Yaskawa INFORM job: X2_99(90,0).JBI

/JOB
//NAME X2_99(90,0)
///FOLDERNAME X2
//POS
///NPOS 440,440,436,13,0,0
///TOOL 0
///POSTYPE PULSE
///PULSE
C00000=2000,-99612,-82443,0,53832,0
C00001=-166393,-132062,-92618,58483,55149,81008
C00002=-157482,-99612,-82443,50725,53832,-76817
C00003=-152781,-96239,-78741,49340,50884,-75750
C00004=-150954,-94792,-77210,48744,49760,-75306
C00005=-150957,-94045,-75225,49281,49201,-75681
C00006=-151067,-94769,-77060,48840,49767,-75375
C00007=-148896,-96259,-77631,48213,48319,-74911
C00008=-154925,-106114,-81211,52368,49780,-77962
C00009=-154976,-104737,-78409,53070,49177,-78455
C00010=-153765,-101609,-77307,52041,49068,-77683
C00011=-154727,-103781,-80113,51957,49998,-77663
C00012=-157482,-99612,-82443,50725,53832,-76817
C00013=-126812,-81448,-90767,9472,77282,-14340
C00014=-120783,-85892,-98127,-47,82159,60
C00015=-120791,-78998,-92147,-45,82022,58
C00016=-120812,-59041,-81112,-38,85486,50
C00017=-120812,-59638,-79752,-38,84341,50
C00018=-120812,-59041,-81112,-38,85486,50
C00019=-120792,-70899,-87175,-45,83124,57
C00020=-120810,-72484,-85548,-40,81307,51
C00021=-120817,-76009,-87202,-37,80512,50
C00022=-120816,-72927,-85752,-37,81205,50
C00023=-120792,-71723,-87920,-45,83159,57
C00024=-120783,-85892,-98127,-47,82159,60
C00025=-120841,-86418,-98444,-30,82084,41
C00026=-120867,-62955,-84955,-21,85839,32
C00027=-120862,-57449,-80347,-23,85833,34
C00028=-120862,-58065,-78999,-24,84687,34
C00029=-120862,-57449,-80347,-23,85833,34
C00030=-120848,-76846,-90076,-28,81853,39
C00031=-120700,-77430,-87681,-72,80079,89
C00032=-120707,-73445,-85814,-70,80978,86
C00033=-120700,-77430,-87681,-72,80079,89
C00034=-120841,-86418,-98444,-30,82084,41
C00035=-120877,-85820,-98106,-19,82183,30
C00036=-120894,-60284,-82721,-14,85837,23
C00037=-120891,-57831,-80469,-15,85712,24
C00038=-120891,-58439,-79117,-15,84567,25
C00039=-120891,-57831,-80469,-15,85712,24
C00040=-120882,-76306,-89742,-18,81925,28
C00041=-120632,-76849,-87581,-92,80316,111
C00042=-120641,-72870,-85708,-89,81208,107
C00043=-120899,-105607,-111704,-13,80383,24
C00044=-120899,-105607,-111704,-13,80383,24
C00045=-120329,-64675,-84682,-181,84785,205
C00046=-120337,-61857,-81845,-179,84488,203
C00047=-120337,-62228,-80870,-179,83698,204
C00048=-120337,-61849,-81865,-179,84506,203
C00049=-120308,-72964,-87409,-188,82206,216
C00050=-112365,-66887,-81837,-2540,82030,2815
C00051=-112466,-65041,-80903,-2509,82400,2777
C00052=-112291,-68228,-82506,-2565,81755,2847
C00053=-88690,-37051,-64863,-22386,100281,29037
C00054=-90338,-32373,-60570,-22143,99643,28585
C00055=-86677,-30127,-56933,-28301,101078,28609
C00056=-87262,-30704,-57322,-28229,100840,28451
C00057=-86036,-30845,-57417,-28365,101220,28810
C00058=-80749,-50154,-73696,-28906,103010,30322
C00059=-106026,-92840,-102541,-4408,81700,4909
C00060=-104933,-21068,-63327,-14588,98299,15445
C00061=-118026,-7058,-59426,2478,121298,42537
C00062=-119206,-9959,-57512,2402,118662,42076
C00063=-119679,-11008,-56668,2374,117617,41892
C00064=-119678,-12040,-55711,2348,116499,41868
C00065=-119679,-11008,-56668,2374,117617,41892
C00066=-117888,-11929,-55575,2351,116426,42475
C00067=-118578,-11982,-55616,2350,116441,42241
C00068=-117888,-11929,-55575,2351,116426,42475
C00069=-116239,-8118,-58416,2447,120087,43116
C00070=-117941,-7017,-59404,2478,121303,42566
C00071=-119121,-9922,-57492,2402,118667,42105
C00072=-119594,-10972,-56650,2375,117622,41921
C00073=-119593,-12004,-55694,2348,116504,41897
C00074=-119594,-10972,-56650,2375,117622,41921
C00075=-117972,-11968,-55595,2351,116420,42446
C00076=-118663,-12020,-55635,2349,116436,42212
C00077=-117972,-11968,-55595,2351,116420,42446
C00078=-116323,-8162,-58441,2447,120082,43087
C00079=-118213,-4464,-57342,2479,121353,42475
C00080=-119375,-7335,-55445,2404,118742,42020
C00081=-119840,-8375,-54609,2376,117706,41839
C00082=-119839,-9401,-53662,2350,116597,41815
C00083=-119840,-8375,-54609,2376,117706,41839
C00084=-117787,-9255,-53494,2353,116516,42511
C00085=-118466,-9310,-53537,2352,116532,42281
C00086=-117787,-9255,-53494,2353,116516,42511
C00087=-113921,-56504,-90793,-659,90254,43086
C00088=-172997,-84117,-74043,29270,60841,12459
C00089=-182497,-62439,-47217,33561,35566,5540
C00090=-177866,51889,12751,25241,78726,20035
C00091=-177567,56483,20827,25353,76270,19609
C00092=-177451,58453,24226,25418,75255,19428
C00093=-177454,58193,25598,25524,74370,19231
C00094=-177460,58244,25401,25510,74505,19259
C00095=-177296,61431,29027,25518,73918,19189
C00096=-177460,58244,25401,25510,74505,19259
C00097=-177875,51523,13769,25307,77989,19872
C00098=-167005,53799,14731,23971,77323,24144
C00099=-166588,57735,22127,23390,74500,23603
C00100=-165356,57001,22663,20748,72181,23241
C00101=-165358,56731,24024,20856,71266,23076
C00102=-165347,56799,23771,20830,71442,23111
C00103=-165330,60004,27398,20889,70889,23018
C00104=-165347,56799,23771,20830,71442,23111
C00105=-166977,49436,12685,24253,74137,23502
C00106=-182364,4853,-37106,25072,86261,16971
C00107=-152303,-102933,-107906,-365,71882,21471
C00108=-90355,-25240,-62492,-31182,91940,-14489
C00109=-138081,35844,8180,-39695,66399,-31141
C00110=-138669,40694,16134,-40133,64268,-30541
C00111=-138897,42750,19469,-40345,63394,-30283
C00112=-138897,42781,21161,-40673,62603,-29947
C00113=-138886,42628,20611,-40593,62809,-30029
C00114=-139201,45623,23796,-40603,62339,-29981
C00115=-138886,42628,20611,-40593,62809,-30029
C00116=-138069,35590,9192,-39905,65818,-30900
C00117=-133067,14417,-5479,-38193,49171,-52584
C00118=-129431,19961,2498,-38515,39991,-63248
C00119=-130261,24926,10174,-39520,37911,-62617
C00120=-130583,27008,13377,-40001,37063,-62330
C00121=-130583,27275,15303,-40912,36255,-61820
C00122=-130584,27314,14967,-40710,36428,-61933
C00123=-131029,30096,17715,-40568,36020,-61996
C00124=-130584,27314,14967,-40710,36428,-61933
C00125=-124769,26347,15261,-56693,39526,-56291
C00126=-125951,31813,23350,-58329,37603,-55322
C00127=-125990,33793,23574,-57346,38066,-55879
C00128=-123661,25065,17775,-59577,38998,-54642
C00129=-125990,34597,27233,-59382,37066,-54726
C00130=-126486,36192,28495,-62823,42923,-46041
C00131=-130207,41845,28467,-57474,57413,-30842
C00132=-133480,44167,26403,-51334,63232,-25301
C00133=-133401,42077,23210,-51024,63850,-25633
C00134=-132439,36745,15005,-50531,65875,-26297
C00135=-90355,-25240,-62492,-31182,91940,-14489
C00136=-126181,-67140,-93758,-13250,84858,5822
C00137=-152303,-102933,-107906,-365,71882,21471
C00138=-151021,-50166,-89002,-846,87371,21807
C00139=-182364,4853,-37106,25072,86261,16971
C00140=-184325,60344,23585,34019,76352,15866
C00141=-183678,65674,32396,34159,73860,15344
C00142=-183957,81689,47427,34502,79595,16153
C00143=-184996,71033,34569,34595,82030,16501
C00144=-183957,81525,49351,34624,78541,15822
C00145=-167608,69842,33487,23377,75298,21262
C00146=-169419,57377,22961,28412,70050,19919
C00147=-169758,52135,14437,28170,72420,20393
C00148=-182364,4853,-37106,25072,86261,16971
C00149=-152303,-102933,-107906,-365,71882,21471
C00150=-121941,-117598,-112997,-12501,69917,32230
C00151=-108451,-171803,-109385,-23800,43994,42320
C00152=-115265,-105280,-99916,-13150,93342,30989
C00153=-112792,-107844,-97393,-16343,91026,32017
C00154=-122694,-143516,-106419,-10106,61697,32034
C00155=-122359,-107950,-95942,-9400,73404,31180
C00156=-122118,-61038,-75540,-9150,84839,30407
C00157=-121770,-8357,-41103,-9216,90729,30109
C00158=-121771,-1968,-35922,-9217,90821,30102
C00159=-121055,-283,-39052,-9429,93653,30116
C00160=-118931,-1420,-16721,-1449,102592,42361
C00161=-118945,163,-15392,-1659,93503,40633
C00162=-120171,930,-10959,-1582,91145,40250
C00163=-120660,1326,-9108,-1553,90200,40098
C00164=-120694,25865,13192,-1550,89085,40100
C00165=-120696,29026,16285,-1550,88805,40104
C00166=-120258,23290,9189,-1576,90234,40233
C00167=-119165,22386,4533,-1644,92655,40570
C00168=-119181,24192,6266,-1459,101602,42286
C00169=-120260,23811,9690,-1517,99280,41943
C00170=-120693,23749,11149,-1541,98342,41806
C00171=-120660,1326,-9108,-1544,99287,41805
C00172=-120174,1432,-10536,-1517,100229,41961
C00173=-118965,1918,-13913,-1451,102579,42349
C00174=-119164,21752,3941,-1459,101779,42290
C00175=-120255,21351,7351,-1518,99456,41942
C00176=-120694,21281,8802,-1542,98518,41803
C00177=-120641,1282,-9371,-1543,99426,41811
C00178=-120163,-1908,-13337,-1516,100237,41964
C00179=-118931,-1420,-16721,-1449,102592,42361
C00180=-109578,15420,-7310,-28367,110236,-41857
C00181=-109763,14188,-4345,-27924,107995,-41350
C00182=-110193,13805,-2890,-27787,106881,-41239
C00183=-131022,13378,-3260,-29129,99839,-47636
C00184=-122106,10683,8881,-53521,92538,-44133
C00185=-120623,10562,7326,-53535,93941,-44154
C00186=-119164,10594,3761,-53715,96134,-44669
C00187=-115308,-32515,-29810,-53374,97452,-43308
C00188=-160324,-56725,-62447,4686,86573,-10750
C00189=-150232,17988,-5017,26557,112251,35280
C00190=-142954,11495,-10959,27504,110227,37702
C00191=-142768,10690,-7556,27067,107926,37200
C00192=-143003,11007,-5424,26849,106972,36875
C00193=-137789,7639,-8393,27391,105376,38540
C00194=-140743,9596,5422,48538,102657,38323
C00195=-145934,20226,29397,62426,105383,26201
C00196=-142397,10029,6905,51885,103476,38119
C00197=-144627,12481,5478,52145,106089,38424
C00198=-150232,17988,-5017,26557,112251,35280
C00199=-160324,-56725,-62447,4686,86573,-10750
C00200=-146496,-53907,-57071,50358,82742,77471
C00201=-142086,-46087,-49611,49702,79955,78251
C00202=-140910,-47839,-49478,49629,78666,78171
C00203=-141016,-46873,-48908,49627,78820,78198
C00204=-140042,-41059,-45363,49344,78825,78701
C00205=-141209,-66264,-43604,72924,53654,56912
C00206=-144414,-64476,-42796,72863,55989,56716
C00207=-142865,-68044,-45540,72856,54877,56844
C00208=-146705,-71229,-49721,72532,57818,56833
C00209=-150615,-73008,-67005,51145,82624,75252
C00210=-84213,-62636,-84550,-16381,94117,81885
C00211=-95245,-30826,-59151,-14149,92862,78402
C00212=-96701,-43295,-61552,-15492,82772,78870
C00213=-98227,-44091,-62190,-15063,82479,78389
C00214=-94037,-41035,-61513,-16198,84364,79567
C00215=-63521,1839,6360,-71273,102323,80160
C00216=-65232,-1066,5117,-71288,100899,80280
C00217=-65232,-364,7293,-71071,100558,80717
C00218=-61873,133,7709,-70638,102845,81131
C00219=-97631,-84017,-82277,-6042,71977,80454
C00220=-97631,-84017,-82277,-6042,71977,13540
C00221=-100992,-100869,-74320,-15072,37892,15545
C00222=-103157,-95187,-70426,-13089,38023,14317
C00223=-103157,-92961,-65713,-13621,36312,14617
C00224=-97699,-120955,-80408,-20799,32327,18909
C00225=2000,-45096,-51939,0,82773,0
C00226=2000,-45096,-51939,0,82773,0
C00227=2000,-45096,-51939,0,82773,0
C00228=2000,-45096,-51939,0,82773,0
C00229=2000,-45096,-51939,0,82773,0
C00230=-70410,-104162,-83449,-55661,60383,81011
C00231=-84923,-92751,-76765,-50721,53081,76684
C00232=-86734,-91468,-75289,-50215,51915,76295
C00233=-86736,-90744,-73307,-50726,51361,76670
C00234=-86623,-91438,-75136,-50303,51925,76361
C00235=-88689,-93063,-75778,-49797,50498,75974
C00236=-86623,-91438,-75136,-50303,51925,76361
C00237=-82499,-102310,-79219,-53526,52313,78845
C00238=-82460,-100986,-76424,-54186,51705,79335
C00239=-83746,-97994,-75341,-53258,51491,78599
C00240=-82460,-100986,-76424,-54186,51705,79335
C00241=-83820,-89231,-90898,-31984,73153,45470
C00242=-103333,-81093,-95821,-5106,83352,5547
C00243=-105734,-58391,-81894,-4383,86302,4664
C00244=-106051,-55558,-79074,-4290,86007,4572
C00245=-106052,-56155,-77720,-4294,84870,4611
C00246=-106051,-55558,-79074,-4290,86007,4572
C00247=-104417,-72181,-87594,-4790,82806,5215
C00248=-104401,-72744,-85473,-4810,81218,5281
C00249=-104801,-68935,-83629,-4684,82015,5119
C00250=-104401,-72744,-85473,-4810,81218,5281
C00251=-103333,-81093,-95821,-5106,83352,5547
C00252=-121034,-86160,-98106,184,81635,-191
C00253=-120937,-60313,-84022,154,86250,-153
C00254=-120931,-57182,-80055,152,85416,-152
C00255=-120931,-57770,-78693,152,84276,-154
C00256=-120931,-57182,-80055,152,85416,-152
C00257=-120995,-76536,-89732,172,81427,-178
C00258=-121142,-77068,-87314,217,79666,-229
C00259=-121124,-73096,-85459,211,80565,-222
C00260=-121142,-77068,-87314,217,79666,-229
C00261=-121096,-115670,-111851,205,74930,-222
C00262=-121096,-115670,-111851,205,74930,-222
C00263=-111920,-77360,-89293,-2569,80863,2809
C00264=-113418,-69208,-82911,-2118,81083,2310
C00265=-113298,-70113,-82134,-2157,80142,2365
C00266=-113298,-69851,-83365,-2151,81033,2349
C00267=-112830,-79068,-87705,-2304,78982,2541
C00268=-118405,-74923,-83336,-614,78322,682
C00269=-118432,-73250,-82545,-605,78695,671
C00270=-118359,-77891,-84712,-629,77644,701
C00271=-147649,-49700,-70143,21952,96038,-28312
C00272=-144092,-44169,-65180,21423,94945,-27268
C00273=-143301,-44665,-65479,21298,94683,-27039
C00274=-145130,-43494,-64769,21581,95292,-27566
C00275=-153783,-86392,-93366,22522,93398,-30972
C00276=-150910,-93017,-97560,17688,85250,-21630
C00277=-120908,-62091,-84868,144,85857,-144
C00278=-120903,-58004,-80414,143,85215,-144
C00279=-120903,-58580,-79044,143,84076,-145
C00280=-120903,-58004,-80414,143,85215,-144
C00281=-120961,-76486,-89626,161,81387,-167
C00282=-121210,-76970,-87437,238,79792,-251
C00283=-121190,-72994,-85579,231,80691,-243
C00284=-121210,-76970,-87437,238,79792,-251
C00285=-120997,-86105,-97999,172,81597,-178
C00286=-122173,-44832,-80249,-1138,103105,-21360
C00287=-123342,-6609,-59067,-2432,120936,-42504
C00288=-122164,-9458,-57119,-2365,118305,-42047
C00289=-121693,-10486,-56262,-2341,117263,-41864
C00290=-121692,-11496,-55292,-2315,116147,-41841
C00291=-121693,-10486,-56262,-2341,117263,-41864
C00292=-123477,-11388,-55156,-2308,116075,-42444
C00293=-122789,-11440,-55197,-2311,116090,-42211
C00294=-123477,-11388,-55156,-2308,116075,-42444
C00295=-125124,-7649,-58044,-2392,119728,-43080
C00296=-123427,-6569,-59045,-2432,120941,-42533
C00297=-122249,-10161,-56477,-2346,117547,-42058
C00298=-121777,-10451,-56245,-2341,117268,-41893
C00299=-121777,-11461,-55275,-2315,116153,-41870
C00300=-121777,-10451,-56245,-2341,117268,-41893
C00301=-123393,-11428,-55177,-2309,116069,-42415
C00302=-122704,-11478,-55216,-2311,116085,-42182
C00303=-123393,-11428,-55177,-2309,116069,-42415
C00304=-123141,-2998,-56146,-2434,120999,-42438
C00305=-121991,-6366,-54527,-2366,118305,-41988
C00306=-121527,-6824,-53376,-2344,117373,-41811
C00307=-121527,-7826,-52419,-2319,116269,-41787
C00308=-121527,-6824,-53376,-2344,117373,-41811
C00309=-123560,-7684,-52253,-2311,116189,-42474
C00310=-122887,-7737,-52295,-2313,116204,-42247
C00311=-123560,-7684,-52253,-2311,116189,-42474
C00312=-125171,-3981,-55094,-2393,119797,-43097
C00313=-101327,-45531,-60072,-2075,102128,-34667
C00314=-89266,4396,-33928,-11465,93507,-29927
C00315=-79229,40490,546,-19170,75952,-25029
C00316=-79192,44826,8093,-19384,73673,-24644
C00317=-79178,46660,11239,-19482,72737,-24484
C00318=-79179,46328,12551,-19579,71812,-24330
C00319=-79171,46385,12358,-19567,71954,-24351
C00320=-79150,49416,15631,-19623,71528,-24272
C00321=-79171,46385,12358,-19567,71954,-24351
C00322=-79222,40075,1538,-19236,75173,-24900
C00323=-94467,40678,813,-12417,73109,-29814
C00324=-94083,44902,8245,-12754,70817,-29441
C00325=-93934,46692,11343,-12898,69876,-29287
C00326=-93935,46363,12659,-12975,68921,-29182
C00327=-93944,46449,12421,-12955,69106,-29206
C00328=-93737,49413,15622,-13089,68702,-29088
C00329=-93944,46449,12421,-12955,69106,-29206
C00330=-94477,40302,1770,-12461,72343,-29738
C00331=-89266,4396,-33928,-11465,93507,-29927
C00332=-101327,-45531,-60072,-2075,102128,-34667
C00333=-154347,-58865,-59313,31959,84488,20300
C00334=-132804,-7309,-34611,38234,83249,26564
C00335=-122368,37716,10148,50470,78338,25854
C00336=-122011,44734,21095,50873,76111,24806
C00337=-122399,46275,23078,51041,76048,24565
C00338=-122399,46336,24666,51210,75440,24220
C00339=-122454,46297,23771,51128,75811,24401
C00340=-121691,49580,27315,51042,75070,24390
C00341=-122454,46284,23500,51099,75914,24459
C00342=-125132,37819,11526,51275,79326,24970
C00343=-124576,6255,-12780,47438,56902,47453
C00344=-122250,19334,1935,46182,44641,59320
C00345=-122250,19334,1935,46182,44641,59320
C00346=-120782,25934,12333,47564,41782,58376
C00347=-120782,26215,14271,48443,41066,57848
C00348=-120776,26249,13930,48246,41217,57966
C00349=-120208,28831,16455,48074,40759,58046
C00350=-120776,26249,13930,48246,41217,57966
C00351=-134725,36017,27474,66792,49610,50401
C00352=-134127,37360,27871,66271,49401,50755
C00353=-134767,35094,27603,67235,49407,50088
C00354=-134127,37993,30581,67335,48840,50017
C00355=-127191,47291,30418,58717,76260,21515
C00356=-128263,40961,20002,56228,76218,21701
C00357=-128172,35801,14205,55931,76570,22030
C00358=-132804,-7309,-34611,38234,83249,26564
C00359=-154347,-58865,-59313,31959,84488,20300
C00360=-101327,-45531,-60072,-2075,102128,-34667
C00361=-89266,4396,-33928,-11465,93507,-29927
C00362=-72391,40299,1753,-27854,73409,-20952
C00363=-72736,45163,9573,-28027,71245,-20542
C00364=-72869,47173,12976,-28133,70261,-20345
C00365=-87821,48907,14678,-21152,65828,-25051
C00366=-88109,46925,11431,-20858,66676,-25318
C00367=-88154,41926,3429,-20512,68875,-25737
C00368=-87331,-25296,-55522,-7683,87670,-26764
C00369=-122814,-32456,-61337,1775,104645,-40589
C00370=-122529,-8270,-43778,1771,106261,-40473
C00371=-133051,-7738,-34192,18720,102488,-41705
C00372=-136275,-43068,-52304,23936,74629,-47166
C00373=-134687,-26689,-41661,23266,75899,-46320
C00374=-131928,8742,-13635,22153,76291,-45269
C00375=-129364,67696,46734,22006,69326,-45649
C00376=-129265,71392,51088,22079,68572,-45758
C00377=-129979,71219,47688,22050,70626,-45633
C00378=-122412,-533,-15942,1476,102193,-42339
C00379=-122403,540,-15029,1679,93098,-40614
C00380=-121179,1356,-10556,1597,90741,-40233
C00381=-120574,1774,-8687,1557,89793,-40041
C00382=-120532,26429,13697,1554,88684,-40039
C00383=-121099,23723,9564,1591,89850,-40218
C00384=-122190,22771,4863,1663,92275,-40553
C00385=-122175,24579,6594,1485,101224,-42269
C00386=-121098,24245,10065,1538,98897,-41927
C00387=-120630,24202,11544,1561,97957,-41779
C00388=-120666,1773,-8688,1564,98883,-41779
C00389=-121177,1858,-10134,1538,99825,-41943
C00390=-122384,2295,-13553,1478,102176,-42330
C00391=-122189,22661,4761,1485,101367,-42272
C00392=-121101,22312,8220,1538,99039,-41927
C00393=-120664,22262,9692,1560,98100,-41789
C00394=-120644,766,-9415,1564,98810,-41771
C00395=-121185,-971,-12517,1537,99838,-41946
C00396=-122412,-533,-15942,1476,102193,-42339
C00397=-131781,15460,-7279,28376,109886,41795
C00398=-131592,14275,-4268,27940,107640,41290
C00399=-131503,14118,-2773,27783,106722,41093
C00400=-110365,13875,-2999,29065,99587,47581
C00401=-120145,11200,9350,53476,92778,43812
C00402=-120732,10849,7590,53521,93669,44023
C00403=-122191,10834,3980,53696,95864,44539
C00404=-128646,-26020,-30624,53883,101032,13133
C00405=-66557,-34885,-48546,-20214,102394,-2504
C00406=-79484,36547,13079,-24373,114005,-30975
C00407=-85904,26694,3247,-25718,112997,-33343
C00408=-86041,25965,6661,-25253,110710,-32858
C00409=-86402,26110,8646,-25107,109560,-32737
C00410=-90488,21267,4070,-25796,108613,-34139
C00411=-88154,25384,22913,-49666,108029,-34753
C00412=-86352,23519,22887,-52150,107314,-32505
C00413=-84237,28413,32993,-57339,108017,-31709
C00414=-87086,25419,21214,-49770,109322,-34894
C00415=-85922,26350,18486,-50250,111381,-35429
C00416=-81578,31234,5255,-15438,110633,-30982
C00417=-71416,-31459,-49219,-37385,106309,-54903
C00418=-79334,-27512,-40554,-52438,93314,-75230
C00419=-81671,-29746,-39165,-52092,90747,-74997
C00420=-82927,-31826,-39398,-51944,89460,-74930
C00421=-82828,-30765,-38686,-51956,89581,-74947
C00422=-84254,-26168,-35546,-51810,89054,-75403
C00423=-79369,-49621,-34755,-72713,68891,-55712
C00424=-83639,-30110,-37749,-52241,83019,-70160
C00425=-77493,-50941,-36554,-72626,70323,-55695
C00426=-74018,-52299,-39928,-72336,73171,-55924
C00427=-60945,-55409,-65093,-53734,104166,-71681
C00428=-60945,-55409,-65093,-53734,104166,-71681
C00429=-127789,-76367,-82464,-10340,71927,-66680
C00430=-126395,-68335,-70990,-10768,62738,-65273
C00431=-128368,-67800,-70596,-9819,62518,-66000
C00432=-129736,-90807,-85563,-9383,59779,-66288
C00433=-134440,-102926,-90239,1517,55386,-10396
C00434=-137693,-99872,-71253,8781,33093,-13294
C00435=-140882,-99069,-62349,23538,21711,-19417
C00436=-140882,-96084,-57211,25293,20222,-20256
C00437=-141874,-99800,-58459,28296,19507,-21772
C00438=-122092,-114409,-88723,8345,70481,-11232
C00439=2000,-48025,-60869,0,102856,0
BC00000=0,666204,302418
BC00001=33147,674408,66891
BC00002=34043,674630,60526
BC00003=34043,674630,60526
BC00004=34043,674630,60526
BC00005=34043,674630,60526
BC00006=34043,674630,60526
BC00007=34043,674630,60526
BC00008=34043,674630,60526
BC00009=34043,674630,60526
BC00010=34043,674630,60526
BC00011=34043,674630,60526
BC00012=34043,674630,60526
BC00013=15644,667481,91364
BC00014=12814,672902,59330
BC00015=12814,672902,59330
BC00016=12814,672902,59330
BC00017=12814,672902,59330
BC00018=12814,672902,59330
BC00019=12814,672902,59330
BC00020=12814,672902,59330
BC00021=12814,672902,59330
BC00022=12814,672902,59330
BC00023=12814,672902,59330
BC00024=12814,672902,59330
BC00025=70623,673655,58742
BC00026=70623,673655,58742
BC00027=70623,673655,58742
BC00028=70623,673655,58742
BC00029=70623,673655,58742
BC00030=70623,673655,58742
BC00031=70623,673655,58742
BC00032=70623,673655,58742
BC00033=70623,673655,58742
BC00034=70623,673655,58742
BC00035=129248,673621,59299
BC00036=129248,673621,59299
BC00037=129248,673621,59299
BC00038=129248,673621,59299
BC00039=129248,673621,59299
BC00040=129248,673621,59299
BC00041=129248,673621,59299
BC00042=129248,673621,59299
BC00043=129248,669709,59299
BC00044=389488,669709,59299
BC00045=389488,669709,59299
BC00046=389488,669709,59299
BC00047=389488,669709,59299
BC00048=389488,669709,59299
BC00049=389488,669709,59299
BC00050=389488,669709,59299
BC00051=389488,669709,59299
BC00052=389488,669709,59299
BC00053=389488,669709,59299
BC00054=389488,669709,59299
BC00055=389488,669709,59299
BC00056=389488,669709,59299
BC00057=389488,669709,59299
BC00058=389488,669709,59299
BC00059=129248,671899,59299
BC00060=129248,671899,59299
BC00061=131979,699465,58241
BC00062=131979,699465,58241
BC00063=131979,699465,58241
BC00064=131979,699465,58241
BC00065=131979,699465,58241
BC00066=131979,699465,58241
BC00067=131979,699465,58241
BC00068=131979,699465,58241
BC00069=131979,699465,58241
BC00070=132002,746034,57968
BC00071=132002,746034,57968
BC00072=132002,746034,57968
BC00073=132002,746034,57968
BC00074=132002,746034,57968
BC00075=132002,746034,57968
BC00076=132002,746034,57968
BC00077=132002,746034,57968
BC00078=132002,746034,57968
BC00079=131294,789553,57813
BC00080=131294,789553,57813
BC00081=131294,789553,57813
BC00082=131294,789553,57813
BC00083=131294,789553,57813
BC00084=131294,789553,57813
BC00085=131294,789553,57813
BC00086=131294,789553,57813
BC00087=131294,789553,57813
BC00088=183654,789553,192797
BC00089=205319,789553,241609
BC00090=192952,789553,63191
BC00091=192952,789553,63191
BC00092=192952,789553,63191
BC00093=192952,789553,63191
BC00094=192952,789553,63191
BC00095=192952,789553,63191
BC00096=192952,789553,63191
BC00097=192952,789553,63191
BC00098=197720,789553,63337
BC00099=197720,789553,63337
BC00100=197720,789553,63337
BC00101=197720,789553,63337
BC00102=197720,789553,63337
BC00103=197720,789553,63337
BC00104=197720,789553,63337
BC00105=197720,789553,63337
BC00106=190214,789553,90491
BC00107=160526,789553,32122
BC00108=129825,789553,81519
BC00109=178627,789553,88525
BC00110=178627,789553,88525
BC00111=178627,789553,88525
BC00112=178627,789553,88525
BC00113=178627,789553,88525
BC00114=178627,789553,88525
BC00115=178627,789553,88525
BC00116=178627,789553,88525
BC00117=173223,789553,85007
BC00118=170379,789553,83156
BC00119=170379,789553,83156
BC00120=170379,789553,83156
BC00121=170379,789553,83156
BC00122=170379,789553,83156
BC00123=170379,789553,83156
BC00124=170379,789553,83156
BC00125=170693,789553,81519
BC00126=170693,789553,81519
BC00127=170693,789553,81519
BC00128=170693,789553,81519
BC00129=170693,789553,81519
BC00130=170693,789553,81518
BC00131=170693,789553,81519
BC00132=170693,789553,81519
BC00133=170693,789553,81519
BC00134=170693,789553,81519
BC00135=129825,789553,81519
BC00136=147580,789553,52951
BC00137=160526,789553,32122
BC00138=160526,789553,32122
BC00139=190214,789553,90491
BC00140=205319,789553,32122
BC00141=205319,789553,32122
BC00142=205319,789553,32122
BC00143=205319,789553,32122
BC00144=205319,789553,32122
BC00145=205319,789553,32122
BC00146=205319,789553,32122
BC00147=205319,789553,32122
BC00148=190214,789553,90491
BC00149=160526,789553,32122
BC00150=160526,789553,32122
BC00151=160526,755651,104205
BC00152=160526,755651,95624
BC00153=160504,755642,95669
BC00154=160504,755642,95669
BC00155=160504,755642,95669
BC00156=160504,755642,95669
BC00157=160473,755492,96017
BC00158=160473,755492,96017
BC00159=160473,755492,96017
BC00160=143735,675447,281889
BC00161=143425,748886,281271
BC00162=143425,748886,281271
BC00163=143425,748886,281271
BC00164=143425,748886,281271
BC00165=143425,748886,281271
BC00166=143425,748886,281271
BC00167=143425,748886,281271
BC00168=143559,719962,281608
BC00169=143559,719962,281608
BC00170=143559,719962,281608
BC00171=143559,719962,281608
BC00172=143559,719962,281608
BC00173=143559,719962,281608
BC00174=143735,675447,281889
BC00175=143735,675447,281889
BC00176=143735,675447,281889
BC00177=143735,675447,281889
BC00178=143735,675447,281889
BC00179=143735,675447,281889
BC00180=146695,666220,221883
BC00181=146695,666220,221883
BC00182=146695,666220,221883
BC00183=146695,666220,221883
BC00184=146695,666220,221881
BC00185=146695,666220,221883
BC00186=146695,666220,221883
BC00187=146695,666220,221883
BC00188=15,666220,224435
BC00189=15,666220,224435
BC00190=15,666220,224435
BC00191=15,666220,224435
BC00192=15,666220,224435
BC00193=15,666220,224435
BC00194=15,666220,224435
BC00195=15,666220,224435
BC00196=15,666220,224435
BC00197=15,666220,224435
BC00198=15,666220,224435
BC00199=15,666220,224435
BC00200=16,666221,121466
BC00201=15,666220,121470
BC00202=15,666220,121470
BC00203=15,666220,121470
BC00204=15,666220,121470
BC00205=15,666220,121470
BC00206=15,666220,121470
BC00207=15,666220,121470
BC00208=15,666220,121470
BC00209=15,666220,121470
BC00210=383087,666220,121470
BC00211=383087,666220,121470
BC00212=383087,666220,121470
BC00213=383087,666220,121470
BC00214=383087,666220,121470
BC00215=383087,666220,121470
BC00216=383087,666220,121470
BC00217=383087,666220,121470
BC00218=383087,666220,121470
BC00219=383087,666220,121470
BC00220=383087,666220,121470
BC00221=383087,666220,121470
BC00222=383087,666220,121470
BC00223=383087,666220,121470
BC00224=383087,666220,121470
BC00225=15,666220,1075229
BC00226=15,666220,1075229
BC00227=15,666220,1075229
BC00228=15,666220,1075229
BC00229=15,666220,1075229
BC00230=398174,675740,57967
BC00231=398174,675740,57967
BC00232=398174,675740,57967
BC00233=398174,675740,57967
BC00234=398174,675740,57967
BC00235=398174,675740,57967
BC00236=398174,675740,57967
BC00237=398174,675740,57967
BC00238=398174,675740,57967
BC00239=398174,675740,57967
BC00240=398174,675740,57967
BC00241=398174,674932,57390
BC00242=398174,674023,56741
BC00243=398174,674023,56741
BC00244=398174,674023,56741
BC00245=398174,674023,56741
BC00246=398174,674023,56741
BC00247=398174,674023,56741
BC00248=398174,674023,56741
BC00249=398174,674023,56741
BC00250=398174,674023,56741
BC00251=398174,674023,56741
BC00252=366924,674754,56144
BC00253=366924,674754,56144
BC00254=366924,674754,56144
BC00255=366924,674754,56144
BC00256=366924,674754,56144
BC00257=366924,674754,56144
BC00258=366924,674754,56144
BC00259=366924,674754,56144
BC00260=366924,674754,56144
BC00261=366924,674754,56144
BC00262=30712,674754,56144
BC00263=30712,674754,68643
BC00264=30712,674754,68643
BC00265=30712,674754,68643
BC00266=30712,674754,68643
BC00267=30712,674754,68643
BC00268=30712,674754,68643
BC00269=30712,674754,68643
BC00270=30712,674754,68643
BC00271=30712,674754,68643
BC00272=30712,674754,68643
BC00273=30712,674754,68643
BC00274=30712,674754,68643
BC00275=30712,674754,68643
BC00276=339116,680642,91140
BC00277=308298,674696,56672
BC00278=308298,674696,56672
BC00279=308298,674696,56672
BC00280=308298,674696,56672
BC00281=308298,674696,56672
BC00282=308298,674696,56672
BC00283=308298,674696,56672
BC00284=308298,674696,56672
BC00285=308298,674696,56672
BC00286=306928,687618,56444
BC00287=305557,700540,56217
BC00288=305557,700540,56217
BC00289=305557,700540,56217
BC00290=305557,700540,56217
BC00291=305557,700540,56217
BC00292=305557,700540,56217
BC00293=305557,700540,56217
BC00294=305557,700540,56217
BC00295=305557,700540,56217
BC00296=305514,747109,57030
BC00297=305514,747109,57030
BC00298=305514,747109,57030
BC00299=305514,747109,57030
BC00300=305514,747109,57030
BC00301=305514,747109,57030
BC00302=305514,747109,57030
BC00303=305514,747109,57030
BC00304=306202,789553,57955
BC00305=306202,789553,57955
BC00306=306202,789553,57955
BC00307=306202,789553,57955
BC00308=306202,789553,57955
BC00309=306202,789553,57955
BC00310=306202,789553,57955
BC00311=306202,789553,57955
BC00312=306202,789553,57955
BC00313=306202,789553,221991
BC00314=298504,779638,136331
BC00315=292117,771411,65252
BC00316=292117,771411,65252
BC00317=292117,771411,65252
BC00318=292117,771411,65252
BC00319=292117,771411,65252
BC00320=292117,771411,65252
BC00321=292117,771411,65252
BC00322=292117,771411,65252
BC00323=297138,774664,65917
BC00324=297138,774664,65917
BC00325=297138,774664,65917
BC00326=297138,774664,65917
BC00327=297138,774664,65917
BC00328=297138,774664,65917
BC00329=297138,774664,65917
BC00330=297138,774664,65917
BC00331=298504,779638,136331
BC00332=306202,789553,221991
BC00333=306202,789553,221991
BC00334=301081,789553,147340
BC00335=309933,789553,80201
BC00336=309933,789553,80201
BC00337=309933,789553,80201
BC00338=309933,789553,80201
BC00339=309933,789553,80201
BC00340=309933,789553,80201
BC00341=309933,789553,80201
BC00342=309933,789553,80201
BC00343=297228,789553,85661
BC00344=297336,789553,84334
BC00345=297336,789553,84334
BC00346=297336,789553,84334
BC00347=297336,789553,84334
BC00348=297336,789553,84334
BC00349=297336,789553,84334
BC00350=297336,789553,84334
BC00351=326204,789553,82063
BC00352=326204,789553,82063
BC00353=326204,789553,82063
BC00354=326204,789553,82063
BC00355=326152,789553,82067
BC00356=326201,789553,82063
BC00357=326204,789553,82063
BC00358=301081,789553,147340
BC00359=306202,789553,221991
BC00360=306202,789553,221991
BC00361=298504,779638,136331
BC00362=283446,773989,34490
BC00363=283446,773989,34490
BC00364=283446,773989,34490
BC00365=283446,773989,34490
BC00366=283446,773989,34490
BC00367=283446,773989,34490
BC00368=288799,761851,159302
BC00369=294036,749978,142630
BC00370=294036,669844,142630
BC00371=294036,669844,142629
BC00372=294036,669844,142629
BC00373=294036,669844,142629
BC00374=294035,670250,143723
BC00375=294034,670267,144116
BC00376=294034,670267,144116
BC00377=294034,670267,144116
BC00378=293812,675994,279822
BC00379=294036,749978,281401
BC00380=294036,749978,281401
BC00381=294036,749978,281401
BC00382=294036,749978,281401
BC00383=294036,749978,281401
BC00384=294036,749978,281401
BC00385=293968,721054,280651
BC00386=293968,721054,280651
BC00387=293968,721054,280651
BC00388=293968,721054,280651
BC00389=293968,721054,280651
BC00390=293968,721054,280651
BC00391=293812,675994,279822
BC00392=293812,675994,279822
BC00393=293812,675994,279822
BC00394=293812,675994,279822
BC00395=293812,675994,279822
BC00396=293812,675994,279822
BC00397=290827,666220,220171
BC00398=290827,666220,220171
BC00399=290827,666220,220171
BC00400=290827,666220,220171
BC00401=290827,666220,220171
BC00402=290827,666220,220171
BC00403=290827,666220,220171
BC00404=290827,666220,220171
BC00405=398174,666220,222117
BC00406=398174,666220,222117
BC00407=398174,666220,222117
BC00408=398174,666220,222117
BC00409=398174,666220,222117
BC00410=398174,666220,222117
BC00411=398174,666220,222117
BC00412=398174,666221,222115
BC00413=398174,666221,222116
BC00414=398174,666220,222117
BC00415=398174,666220,222117
BC00416=398174,666220,222117
BC00417=398174,666220,160700
BC00418=398174,666220,116225
BC00419=398174,666220,116225
BC00420=398174,666220,116225
BC00421=398174,666220,116225
BC00422=398174,666220,116225
BC00423=398174,666220,116225
BC00424=398174,666220,116225
BC00425=398174,666220,116225
BC00426=398174,666220,116225
BC00427=398174,666220,116225
BC00428=59154,666220,116225
BC00429=59154,666220,116225
BC00430=59154,666220,116225
BC00431=59154,666220,116225
BC00432=59154,666220,116225
BC00433=59154,666220,116225
BC00434=59154,666220,116225
BC00435=59154,666220,116221
BC00436=59154,666220,116221
BC00437=59154,666220,116221
BC00438=66146,666218,182566
BC00439=118464,666204,678996
EC00000=798156,0
EC00001=798156,0
EC00002=798156,0
EC00003=798156,0
EC00004=798156,0
EC00005=798156,0
EC00006=798156,0
EC00007=798156,0
EC00008=798156,0
EC00009=798156,0
EC00010=798156,0
EC00011=798156,0
EC00012=798156,0
EC00013=798156,0
EC00014=798156,0
EC00015=798156,0
EC00016=798156,0
EC00017=798156,0
EC00018=798156,0
EC00019=798156,0
EC00020=798156,0
EC00021=798156,0
EC00022=798156,0
EC00023=798156,0
EC00024=798156,0
EC00025=798156,0
EC00026=798156,0
EC00027=798156,0
EC00028=798156,0
EC00029=798156,0
EC00030=798156,0
EC00031=798156,0
EC00032=798156,0
EC00033=798156,0
EC00034=798156,0
EC00035=798156,0
EC00036=798156,0
EC00037=798156,0
EC00038=798156,0
EC00039=798156,0
EC00040=798156,0
EC00041=798156,0
EC00042=798156,0
EC00043=798156,0
EC00044=798156,0
EC00045=798156,0
EC00046=798156,0
EC00047=798156,0
EC00048=798156,0
EC00049=798156,0
EC00050=798156,0
EC00051=798156,0
EC00052=798156,0
EC00053=798156,0
EC00054=798156,0
EC00055=798156,0
EC00056=798156,0
EC00057=798156,0
EC00058=798156,0
EC00059=798156,0
EC00060=798156,0
EC00061=798156,0
EC00062=798156,0
EC00063=798156,0
EC00064=798156,0
EC00065=798156,0
EC00066=798156,0
EC00067=798156,0
EC00068=798156,0
EC00069=798156,0
EC00070=798156,0
EC00071=798156,0
EC00072=798156,0
EC00073=798156,0
EC00074=798156,0
EC00075=798156,0
EC00076=798156,0
EC00077=798156,0
EC00078=798156,0
EC00079=798156,0
EC00080=798156,0
EC00081=798156,0
EC00082=798156,0
EC00083=798156,0
EC00084=798156,0
EC00085=798156,0
EC00086=798156,0
EC00087=798156,0
EC00088=798156,0
EC00089=798156,0
EC00090=798156,0
EC00091=798156,0
EC00092=798156,0
EC00093=798156,0
EC00094=798156,0
EC00095=798156,0
EC00096=798156,0
EC00097=798156,0
EC00098=798156,0
EC00099=798156,0
EC00100=798156,0
EC00101=798156,0
EC00102=798156,0
EC00103=798156,0
EC00104=798156,0
EC00105=798156,0
EC00106=798156,0
EC00107=798156,0
EC00108=798156,0
EC00109=798156,0
EC00110=798156,0
EC00111=798156,0
EC00112=798156,0
EC00113=798156,0
EC00114=798156,0
EC00115=798156,0
EC00116=798156,0
EC00117=798156,0
EC00118=798156,0
EC00119=798156,0
EC00120=798156,0
EC00121=798156,0
EC00122=798156,0
EC00123=798156,0
EC00124=798156,0
EC00125=798156,0
EC00126=798156,0
EC00127=798156,0
EC00128=798155,1
EC00129=798156,0
EC00130=798156,0
EC00131=798156,0
EC00132=798156,0
EC00133=798156,0
EC00134=798156,0
EC00135=798156,0
EC00136=798156,0
EC00137=798156,0
EC00138=798156,0
EC00139=798156,0
EC00140=798156,0
EC00141=798156,0
EC00142=798156,0
EC00143=798156,0
EC00144=798156,0
EC00145=798156,0
EC00146=798156,0
EC00147=798156,0
EC00148=798156,0
EC00149=798156,0
EC00150=798156,0
EC00151=798156,0
EC00152=798156,0
EC00153=798156,0
EC00154=798156,0
EC00155=798156,0
EC00156=798156,0
EC00157=798156,0
EC00158=798156,0
EC00159=798156,0
EC00160=798156,0
EC00161=798156,0
EC00162=798156,0
EC00163=798156,0
EC00164=798156,0
EC00165=798156,0
EC00166=798156,0
EC00167=798156,0
EC00168=798156,0
EC00169=798156,0
EC00170=798156,0
EC00171=798156,0
EC00172=798156,0
EC00173=798156,0
EC00174=798156,0
EC00175=798156,0
EC00176=798156,0
EC00177=798156,0
EC00178=798156,0
EC00179=798156,0
EC00180=798155,1
EC00181=798156,0
EC00182=798156,0
EC00183=798156,0
EC00184=798156,0
EC00185=798156,0
EC00186=798156,0
EC00187=798156,0
EC00188=798156,0
EC00189=798156,0
EC00190=798156,0
EC00191=798156,0
EC00192=798156,0
EC00193=798156,0
EC00194=798156,0
EC00195=798156,0
EC00196=798155,0
EC00197=798156,0
EC00198=798156,0
EC00199=798156,0
EC00200=798156,0
EC00201=798156,0
EC00202=798156,0
EC00203=798156,0
EC00204=798156,0
EC00205=798156,0
EC00206=798156,0
EC00207=798156,0
EC00208=798156,0
EC00209=798156,0
EC00210=798156,0
EC00211=798156,0
EC00212=798156,0
EC00213=798156,0
EC00214=798156,0
EC00215=798156,0
EC00216=798156,0
EC00217=798156,0
EC00218=798156,0
EC00219=798156,0
EC00220=798156,0
EC00221=798156,0
EC00222=310394,0
EC00223=310394,556475
EC00224=310394,1112951
EC00225=798156,1112951
EC00226=798156,1112951
EC00227=798156,1112951
EC00228=798156,1112951
EC00229=798156,1112951
EC00230=798156,1112951
EC00231=798156,1112951
EC00232=798156,1112951
EC00233=798156,1112951
EC00234=798156,1112951
EC00235=798156,1112951
EC00236=798156,1112951
EC00237=798156,1112951
EC00238=798156,1112951
EC00239=798156,1112951
EC00240=798156,1112951
EC00241=798156,1112951
EC00242=798156,1112951
EC00243=798156,1112951
EC00244=798156,1112951
EC00245=798156,1112951
EC00246=798156,1112951
EC00247=798156,1112951
EC00248=798156,1112951
EC00249=798156,1112951
EC00250=798156,1112951
EC00251=798156,1112951
EC00252=798156,1112951
EC00253=798156,1112951
EC00254=798156,1112951
EC00255=798156,1112951
EC00256=798156,1112951
EC00257=798156,1112951
EC00258=798156,1112951
EC00259=798156,1112951
EC00260=798156,1112951
EC00261=798156,1112951
EC00262=798156,1112951
EC00263=798156,1112951
EC00264=798156,1112951
EC00265=798156,1112951
EC00266=798156,1112951
EC00267=798156,1112951
EC00268=798156,1112951
EC00269=798156,1112951
EC00270=798156,1112951
EC00271=798156,1112951
EC00272=798156,1112951
EC00273=798156,1112951
EC00274=798156,1112951
EC00275=798156,1112951
EC00276=798156,1112951
EC00277=798156,1112951
EC00278=798156,1112951
EC00279=798156,1112951
EC00280=798156,1112951
EC00281=798156,1112951
EC00282=798156,1112951
EC00283=798156,1112951
EC00284=798156,1112951
EC00285=798156,1112951
EC00286=798156,1112951
EC00287=798156,1112951
EC00288=798156,1112951
EC00289=798156,1112951
EC00290=798156,1112951
EC00291=798156,1112951
EC00292=798156,1112951
EC00293=798156,1112951
EC00294=798156,1112951
EC00295=798156,1112951
EC00296=798156,1112951
EC00297=798156,1112951
EC00298=798156,1112951
EC00299=798156,1112951
EC00300=798156,1112951
EC00301=798156,1112951
EC00302=798156,1112951
EC00303=798156,1112951
EC00304=798156,1112951
EC00305=798156,1112951
EC00306=798156,1112951
EC00307=798156,1112951
EC00308=798156,1112951
EC00309=798156,1112951
EC00310=798156,1112951
EC00311=798156,1112951
EC00312=798156,1112951
EC00313=798156,1112951
EC00314=798156,1112951
EC00315=798156,1112951
EC00316=798156,1112951
EC00317=798156,1112951
EC00318=798156,1112951
EC00319=798156,1112951
EC00320=798156,1112951
EC00321=798156,1112951
EC00322=798156,1112951
EC00323=798156,1112951
EC00324=798156,1112951
EC00325=798156,1112951
EC00326=798156,1112951
EC00327=798156,1112951
EC00328=798156,1112951
EC00329=798156,1112951
EC00330=798156,1112951
EC00331=798156,1112951
EC00332=798156,1112951
EC00333=798156,1112951
EC00334=798156,1112951
EC00335=798156,1112951
EC00336=798156,1112951
EC00337=798156,1112951
EC00338=798156,1112951
EC00339=798156,1112951
EC00340=798156,1112951
EC00341=798156,1112951
EC00342=798156,1112951
EC00343=798156,1112951
EC00344=798156,1112951
EC00345=798156,1112951
EC00346=798156,1112951
EC00347=798156,1112951
EC00348=798156,1112951
EC00349=798156,1112951
EC00350=798156,1112951
EC00351=798156,1112951
EC00352=798156,1112951
EC00353=798156,1112951
EC00354=798156,1112951
EC00355=798156,1112951
EC00356=798156,1112951
EC00357=798156,1112951
EC00358=798156,1112951
EC00359=798156,1112951
EC00360=798156,1112951
EC00361=798156,1112951
EC00362=798156,1112951
EC00363=798156,1112951
EC00364=798156,1112951
EC00365=798156,1112951
EC00366=798156,1112951
EC00367=798155,1112950
EC00368=798155,1112950
EC00369=798155,1112950
EC00370=798155,1112950
EC00371=798155,1112950
EC00372=798155,1112950
EC00373=798155,1112950
EC00374=798156,1112951
EC00375=798156,1112951
EC00376=798156,1112951
EC00377=798156,1112951
EC00378=798156,1112951
EC00379=798156,1112951
EC00380=798156,1112951
EC00381=798156,1112951
EC00382=798156,1112951
EC00383=798156,1112951
EC00384=798156,1112951
EC00385=798156,1112951
EC00386=798156,1112951
EC00387=798156,1112951
EC00388=798156,1112951
EC00389=798156,1112951
EC00390=798156,1112951
EC00391=798156,1112951
EC00392=798156,1112951
EC00393=798156,1112951
EC00394=798156,1112951
EC00395=798156,1112951
EC00396=798156,1112951
EC00397=798156,1112951
EC00398=798156,1112951
EC00399=798156,1112951
EC00400=798156,1112951
EC00401=798156,1112951
EC00402=798156,1112951
EC00403=798156,1112951
EC00404=798156,1112951
EC00405=798156,1112951
EC00406=798156,1112951
EC00407=798156,1112951
EC00408=798155,1112950
EC00409=798155,1112950
EC00410=798156,1112951
EC00411=798156,1112951
EC00412=798156,1112951
EC00413=798156,1112951
EC00414=798156,1112951
EC00415=798156,1112951
EC00416=798156,1112951
EC00417=798156,1112951
EC00418=798156,1112951
EC00419=798156,1112951
EC00420=798156,1112951
EC00421=798156,1112951
EC00422=798156,1112951
EC00423=798156,1112951
EC00424=798156,1112951
EC00425=798156,1112951
EC00426=798156,1112951
EC00427=798156,1112951
EC00428=798156,1112951
EC00429=798156,1112951
EC00430=798156,1112951
EC00431=798155,1112950
EC00432=798155,1112950
EC00433=798155,1112950
EC00434=798154,1112948
EC00435=798156,1112951
///POSTYPE BASE
///RECTAN
///RCONF 0,0,0,0,0,0,0,0,0,0,0,0,0,0,0,0,0,0,0,0,0,0,0,0
P00006=0.222,-3.123,-1.508,0.0000,0.0000,0.0000
P00021=-0.225,-6.128,-0.405,0.0000,0.0000,0.0000
P00022=0.222,-3.123,-1.508,0.0000,0.0000,0.0000
P00023=0.143,-0.036,0.682,0.0000,0.0000,0.0000
P00024=0.145,-0.552,1.326,0.0000,0.0000,0.0000
P00025=-2.003,0.006,0.728,0.0000,0.0000,0.0000
P00026=0.562,-0.002,-0.337,0.0000,0.0000,0.0000
P00027=-0.746,0.015,-9.096,0.0000,0.0000,0.0000
P00028=-2.237,-0.018,-7.702,0.0000,0.0000,0.0000
P00029=-2.156,-0.086,-4.681,0.0000,0.0000,0.0000
P00030=5.926,-4.294,-1.390,0.0000,0.0000,0.0000
P00031=1.853,-0.001,-1.549,0.0000,0.0000,0.0000
P00045=-0.068,-0.810,1.603,0.0000,0.0000,0.0000
//INST
///DATE 2025/04/14 14:44
///ATTR SC,RW
///GROUP1 RB1,BS1
///GROUP2 ST1
NOP
'X2_99(90,0)
MOVJ C00000 BC00000 VJ=100.00  +MOVJ EC00000 VJ=100.00
MOVJ C00001 BC00001 VJ=100.00  +MOVJ EC00001 VJ=100.00
'Path S4826
SFTOF3D
MOVJ C00002 BC00002 VJ=100.00  +MOVJ EC00002 VJ=100.00
MOVL C00003 BC00003 V=800.0  +MOVJ EC00003 VJ=100.00
SMOVL C00004 BC00004 V=166.7  +MOVJ EC00004
SREFP 3 C00005 BC00005  +REFP EC00005
CALL JOB:SEARCH-R1-S13D
SET P031 P006
SFTON3D P031
SMOVL C00006 BC00006 V=166.7  +MOVJ EC00006
SREFP 3 C00007 BC00007  +REFP EC00007
CALL JOB:SEARCH-R1-S13D
SET P031 P006
SFTON3D P031
SMOVL C00008 BC00008 V=250.0  +MOVJ EC00008
SMOVL C00009 BC00009 V=250.0  +MOVJ EC00009
SREFP 3 C00010 BC00010  +REFP EC00010
CALL JOB:SEARCH-R1-S13D
SET P031 P006
SFTON3D P031
SMOVL C00011 BC00011 V=250.0  +MOVJ EC00011
MOVL C00012 BC00012 V=1000.0  +MOVJ EC00012 VJ=100.00
'EndPath S4826
MOVJ C00013 BC00013 VJ=100.00  +MOVJ EC00013 VJ=100.00
'Path S4869
SFTOF3D
MOVJ C00014 BC00014 VJ=100.00  +MOVJ EC00014 VJ=100.00
MOVL C00015 BC00015 V=800.0  +MOVJ EC00015 VJ=100.00
SMOVL C00016 BC00016 V=250.0  +MOVJ EC00016
SREFP 3 C00017 BC00017  +REFP EC00017
CALL JOB:SEARCH-R1-S13D
SET P030 P006
SFTON3D P030
SMOVL C00018 BC00018 V=166.7  +MOVJ EC00018
SMOVL C00019 BC00019 V=250.0  +MOVJ EC00019
SMOVL C00020 BC00020 V=250.0  +MOVJ EC00020
SMOVL C00021 BC00021 V=166.7  +MOVJ EC00021
SREFP 3 C00022 BC00022  +REFP EC00022
CALL JOB:SEARCH-R1-S13D
SET P030 P006
SFTON3D P030
SMOVL C00023 BC00023 V=250.0  +MOVJ EC00023
MOVL C00024 BC00024 V=1000.0  +MOVJ EC00024 VJ=100.00
'EndPath S4869
'Path S4870
SFTOF3D
MOVJ C00025 BC00025 VJ=100.00  +MOVJ EC00025 VJ=100.00
SMOVL C00026 BC00026 V=1000.0  +MOVJ EC00026
SMOVL C00027 BC00027 V=250.0  +MOVJ EC00027
SREFP 3 C00028 BC00028  +REFP EC00028
CALL JOB:SEARCH-R1-S13D
SET P029 P006
SFTON3D P029
SMOVL C00029 BC00029 V=250.0  +MOVJ EC00029
SMOVL C00030 BC00030 V=1000.0  +MOVJ EC00030
SMOVL C00031 BC00031 V=250.0  +MOVJ EC00031
SREFP 3 C00032 BC00032  +REFP EC00032
CALL JOB:SEARCH-R1-S13D
SET P029 P006
SFTON3D P029
SMOVL C00033 BC00033 V=250.0  +MOVJ EC00033
MOVL C00034 BC00034 V=1000.0  +MOVJ EC00034 VJ=100.00
'EndPath S4870
'Path S4823
SFTOF3D
MOVJ C00035 BC00035 VJ=100.00  +MOVJ EC00035 VJ=100.00
SMOVL C00036 BC00036 V=1000.0  +MOVJ EC00036
SMOVL C00037 BC00037 V=166.7  +MOVJ EC00037
SREFP 3 C00038 BC00038  +REFP EC00038
CALL JOB:SEARCH-R1-S13D
SET P028 P006
SFTON3D P028
SMOVL C00039 BC00039 V=250.0  +MOVJ EC00039
SMOVL C00040 BC00040 V=250.0  +MOVJ EC00040
SMOVL C00041 BC00041 V=250.0  +MOVJ EC00041
SREFP 3 C00042 BC00042  +REFP EC00042
CALL JOB:SEARCH-R1-S13D
SET P028 P006
SFTON3D P028
MOVL C00043 BC00043 V=1000.0  +MOVJ EC00043 VJ=100.00
SFTOF3D
SMOVL C00044 BC00044 V=1200.0  +MOVJ EC00044
SMOVL C00045 BC00045 V=1200.0  +MOVJ EC00045
SMOVL C00046 BC00046 V=166.7  +MOVJ EC00046
SREFP 3 C00047 BC00047  +REFP EC00047
CALL JOB:SEARCH-R1-S13D
SET P045 P006
SFTON3D P045
SMOVL C00048 BC00048 V=166.7  +MOVJ EC00048
SMOVL C00049 BC00049 V=800.0  +MOVJ EC00049
SMOVL C00050 BC00050 V=166.7  +MOVJ EC00050
SREFP 3 C00051 BC00051  +REFP EC00051
CALL JOB:SEARCH-R1-S13D
SET P045 P006
SFTON3D P045
SMOVL C00052 BC00052 V=166.7  +MOVJ EC00052
SMOVL C00053 BC00053 V=800.0  +MOVJ EC00053
SMOVL C00054 BC00054 V=800.0  +MOVJ EC00054
SMOVL C00055 BC00055 V=166.7  +MOVJ EC00055
SREFP 3 C00056 BC00056  +REFP EC00056
CALL JOB:SEARCH-R1-S13D
SET P045 P006
SFTON3D P045
SMOVL C00057 BC00057 V=250.0  +MOVJ EC00057
SMOVL C00058 BC00058 V=1200.0  +MOVJ EC00058
SFTOF3D
SMOVL C00059 BC00059 V=1200.0  +MOVJ EC00059
SMOVL C00060 BC00060 V=1200.0  +MOVJ EC00060
'EndPath S4823
'Path S4871
SFTOF3D
MOVJ C00061 BC00061 VJ=100.00  +MOVJ EC00061 VJ=100.00
MOVL C00062 BC00062 V=500.0  +MOVJ EC00062 VJ=100.00
SMOVL C00063 BC00063 V=166.7  +MOVJ EC00063
SREFP 3 C00064 BC00064  +REFP EC00064
CALL JOB:SEARCH-R1-S13D
SET P027 P006
SFTON3D P027
SMOVL C00065 BC00065 V=250.0  +MOVJ EC00065
SMOVL C00066 BC00066 V=166.7  +MOVJ EC00066
SREFP 3 C00067 BC00067  +REFP EC00067
CALL JOB:SEARCH-R1-S13D
SET P027 P006
SFTON3D P027
SMOVL C00068 BC00068 V=250.0  +MOVJ EC00068
MOVL C00069 BC00069 V=1000.0  +MOVJ EC00069 VJ=100.00
'EndPath S4871
'Path S4872
SFTOF3D
MOVJ C00070 BC00070 VJ=100.00  +MOVJ EC00070 VJ=100.00
MOVL C00071 BC00071 V=500.0  +MOVJ EC00071 VJ=100.00
SMOVL C00072 BC00072 V=166.7  +MOVJ EC00072
SREFP 3 C00073 BC00073  +REFP EC00073
CALL JOB:SEARCH-R1-S13D
SET P026 P006
SFTON3D P026
SMOVL C00074 BC00074 V=250.0  +MOVJ EC00074
SMOVL C00075 BC00075 V=166.7  +MOVJ EC00075
SREFP 3 C00076 BC00076  +REFP EC00076
CALL JOB:SEARCH-R1-S13D
SET P026 P006
SFTON3D P026
SMOVL C00077 BC00077 V=800.0  +MOVJ EC00077
MOVL C00078 BC00078 V=1000.0  +MOVJ EC00078 VJ=100.00
'EndPath S4872
'Path S4820
SFTOF3D
MOVJ C00079 BC00079 VJ=100.00  +MOVJ EC00079 VJ=100.00
MOVL C00080 BC00080 V=500.0  +MOVJ EC00080 VJ=100.00
SMOVL C00081 BC00081 V=166.7  +MOVJ EC00081
SREFP 3 C00082 BC00082  +REFP EC00082
CALL JOB:SEARCH-R1-S13D
SET P025 P006
SFTON3D P025
SMOVL C00083 BC00083 V=250.0  +MOVJ EC00083
SMOVL C00084 BC00084 V=166.7  +MOVJ EC00084
SREFP 3 C00085 BC00085  +REFP EC00085
CALL JOB:SEARCH-R1-S13D
SET P025 P006
SFTON3D P025
SMOVL C00086 BC00086 V=250.0  +MOVJ EC00086
MOVL C00087 BC00087 V=1000.0  +MOVJ EC00087 VJ=100.00
'EndPath S4820
MOVJ C00088 BC00088 VJ=100.00  +MOVJ EC00088 VJ=100.00
MOVJ C00089 BC00089 VJ=100.00  +MOVJ EC00089 VJ=100.00
'Path S4819 (for W4811)
SFTOF3D
MOVJ C00090 BC00090 VJ=100.00  +MOVJ EC00090 VJ=100.00
MOVL C00091 BC00091 V=666.7  +MOVJ EC00091 VJ=100.00
SMOVL C00092 BC00092 V=166.7  +MOVJ EC00092
SREFP 3 C00093 BC00093  +REFP EC00093
CALL JOB:SEARCH-R1-S13D
SET P024 P006
SFTON3D P024
SMOVL C00094 BC00094 V=166.7  +MOVJ EC00094
SREFP 3 C00095 BC00095  +REFP EC00095
CALL JOB:SEARCH-R1-S13D
SET P024 P006
SFTON3D P024
SMOVL C00096 BC00096 V=166.7  +MOVJ EC00096
MOVL C00097 BC00097 V=1000.0  +MOVJ EC00097 VJ=100.00
'EndPath S4819 (for W4811)
'Path S4818 (for W4811)
SFTOF3D
MOVJ C00098 BC00098 VJ=100.00  +MOVJ EC00098 VJ=100.00
MOVL C00099 BC00099 V=500.0  +MOVJ EC00099 VJ=100.00
SMOVL C00100 BC00100 V=166.7  +MOVJ EC00100
SREFP 3 C00101 BC00101  +REFP EC00101
CALL JOB:SEARCH-R1-S13D
SET P023 P006
SFTON3D P023
SMOVL C00102 BC00102 V=166.7  +MOVJ EC00102
SREFP 3 C00103 BC00103  +REFP EC00103
CALL JOB:SEARCH-R1-S13D
SET P023 P006
SFTON3D P023
SMOVL C00104 BC00104 V=166.7  +MOVJ EC00104
MOVL C00105 BC00105 V=1000.0  +MOVJ EC00105 VJ=100.00
'EndPath S4818 (for W4811)
MOVJ C00106 BC00106 VJ=100.00  +MOVJ EC00106 VJ=100.00
MOVJ C00107 BC00107 VJ=100.00  +MOVJ EC00107 VJ=100.00
MOVJ C00108 BC00108 VJ=100.00  +MOVJ EC00108 VJ=100.00
'Path S4816 (for W4808)
SFTOF3D
MOVJ C00109 BC00109 VJ=100.00  +MOVJ EC00109 VJ=100.00
MOVL C00110 BC00110 V=500.0  +MOVJ EC00110 VJ=100.00
SMOVL C00111 BC00111 V=166.7  +MOVJ EC00111
SREFP 3 C00112 BC00112  +REFP EC00112
CALL JOB:SEARCH-R1-S13D
SET P021 P006
SFTON3D P021
SMOVL C00113 BC00113 V=166.7  +MOVJ EC00113
SREFP 3 C00114 BC00114  +REFP EC00114
CALL JOB:SEARCH-R1-S13D
SET P021 P006
SFTON3D P021
SMOVL C00115 BC00115 V=166.7  +MOVJ EC00115
MOVL C00116 BC00116 V=1000.0  +MOVJ EC00116 VJ=100.00
'EndPath S4816 (for W4808)
MOVJ C00117 BC00117 VJ=100.00  +MOVJ EC00117 VJ=100.00
'Path S4817 (for W4808)
SFTOF3D
MOVJ C00118 BC00118 VJ=100.00  +MOVJ EC00118 VJ=100.00
MOVL C00119 BC00119 V=500.0  +MOVJ EC00119 VJ=100.00
SMOVL C00120 BC00120 V=166.7  +MOVJ EC00120
SREFP 3 C00121 BC00121  +REFP EC00121
CALL JOB:SEARCH-R1-S13D
SET P022 P006
SFTON3D P022
SMOVL C00122 BC00122 V=166.7  +MOVJ EC00122
SREFP 3 C00123 BC00123  +REFP EC00123
CALL JOB:SEARCH-R1-S13D
SET P022 P006
SFTON3D P022
SMOVL C00124 BC00124 V=166.7  +MOVJ EC00124
'EndPath S4817 (for W4808)
'Path W4808
SFTOF3D
SFTON3D P022
MOVJ C00125 BC00125 VJ=100.00  +MOVJ EC00125 VJ=100.00
SMOVL C00126 BC00126 V=800.0  +MOVJ EC00126
REFP 1 RB1 C00127 BC00127
REFP 1 RB1 C00128 BC00128
SMOVL C00129 BC00129 V=150.0 PL=0  +MOVJ EC00127
SWVON WEV#(100)
MACRO1 MJ#(0) ARGF21
ARCON
SMOVL C00130 BC00130 V=8.3  +MOVJ EC00128
SFTON3D P021
SMOVL C00131 BC00131 V=8.3  +MOVJ EC00129
SMOVL C00132 BC00132 V=8.3  +MOVJ EC00130
ARCOF
SWVOF
SMOVL C00133 BC00133 V=800.0  +MOVJ EC00131
SMOVL C00134 BC00134 V=1000.0  +MOVJ EC00132
SFTOF3D
'EndPath W4808
MOVJ C00135 BC00135 VJ=100.00  +MOVJ EC00133 VJ=100.00
MOVJ C00136 BC00136 VJ=100.00  +MOVJ EC00134 VJ=100.00
MOVJ C00137 BC00137 VJ=100.00  +MOVJ EC00135 VJ=100.00
MOVJ C00138 BC00138 VJ=100.00  +MOVJ EC00136 VJ=100.00
MOVJ C00139 BC00139 VJ=100.00  +MOVJ EC00137 VJ=100.00
'Path W4811
SFTOF3D
SFTON3D P024
MOVJ C00140 BC00140 VJ=100.00  +MOVJ EC00138 VJ=100.00
SMOVL C00141 BC00141 V=800.0  +MOVJ EC00139
REFP 1 RB1 C00142 BC00142
REFP 2 RB1 C00143 BC00143
SMOVL C00144 BC00144 V=150.0 PL=0  +MOVJ EC00140
MACRO1 MJ#(0) ARGF9
SWVON WEV#(100)
ARCON
SFTON3D P023
SMOVL C00145 BC00145 V=8.3  +MOVJ EC00141
ARCOF
SWVOF
SMOVL C00146 BC00146 V=800.0  +MOVJ EC00142
SMOVL C00147 BC00147 V=1000.0  +MOVJ EC00143
SFTOF3D
'EndPath W4811
'
MOVJ C00148 BC00148 VJ=100.00  +MOVJ EC00144 VJ=100.00
MOVJ C00149 BC00149 VJ=100.00  +MOVJ EC00145 VJ=100.00
MOVJ C00150 BC00150 VJ=100.00  +MOVJ EC00146 VJ=100.00
'Path W4873
SFTOF3D
SFTON3D P027
MOVJ C00151 BC00151 VJ=100.00  +MOVJ EC00147 VJ=100.00
SMOVL C00152 BC00152 V=800.0  +MOVJ EC00148
SMOVL C00153 BC00153 V=150.0 PL=0  +MOVJ EC00149
MACRO1 MJ#(0) ARGF14
ARCON
SMOVL C00154 BC00154 V=10.0  +MOVJ EC00150
SMOVL C00155 BC00155 V=10.8  +MOVJ EC00151
SFTON3D P026
SMOVL C00156 BC00156 V=10.8  +MOVJ EC00152
SFTON3D P025
SMOVL C00157 BC00157 V=10.8  +MOVJ EC00153
MOVL C00158 BC00158 V=10.8  +MOVJ EC00154 VJ=0.78
ARCOF
SMOVL C00159 BC00159 V=800.0  +MOVJ EC00155
SMOVL C00160 BC00160 V=1000.0  +MOVJ EC00156
SFTOF3D
COMM SFTON3D P025
COMM MOVJ C00161 BC00161 VJ=100.00  +MOVJ EC00157 VJ=100.00
COMM SMOVL C00162 BC00162 V=800.0  +MOVJ EC00158
COMM SMOVL C00163 BC00163 V=150.0 PL=0  +MOVJ EC00159
COMM MACRO1 MJ#(0) ARGF14
COMM ARCON
COMM SMOVL C00164 BC00164 V=10.8  +MOVJ EC00160
COMM ARCON
COMM SMOVL C00165 BC00165 V=10.0  +MOVJ EC00161
COMM ARCOF
COMM SMOVL C00166 BC00166 V=800.0  +MOVJ EC00162
COMM SMOVL C00167 BC00167 V=1000.0  +MOVJ EC00163
COMM SFTOF3D
COMM 'EndPath W4873
COMM 'Path W4874
COMM SFTOF3D
COMM SFTON3D P026
COMM MOVJ C00168 BC00168 VJ=100.00  +MOVJ EC00164 VJ=100.00
COMM SMOVL C00169 BC00169 V=800.0  +MOVJ EC00165
COMM SMOVL C00170 BC00170 V=150.0 PL=0  +MOVJ EC00166
COMM ARCON
COMM SMOVL C00171 BC00171 V=10.8  +MOVJ EC00167
COMM ARCOF
COMM SMOVL C00172 BC00172 V=800.0  +MOVJ EC00168
COMM SMOVL C00173 BC00173 V=1000.0  +MOVJ EC00169
COMM SFTOF3D
COMM 'EndPath W4874
COMM 'Path W4875
COMM SFTOF3D
COMM SFTON3D P027
COMM MOVJ C00174 BC00174 VJ=100.00  +MOVJ EC00170 VJ=100.00
COMM SMOVL C00175 BC00175 V=800.0  +MOVJ EC00171
COMM SMOVL C00176 BC00176 V=150.0 PL=0  +MOVJ EC00172
COMM ARCON
COMM SMOVL C00177 BC00177 V=10.8  +MOVJ EC00173
COMM ARCOF
COMM SMOVL C00178 BC00178 V=800.0  +MOVJ EC00174
COMM SMOVL C00179 BC00179 V=1000.0  +MOVJ EC00175
COMM SFTOF3D
'EndPath W4875
'Path W4876
SFTOF3D
SFTON3D P028
MOVJ C00180 BC00180 VJ=100.00  +MOVJ EC00176 VJ=100.00
SMOVL C00181 BC00181 V=800.0  +MOVJ EC00177
SMOVL C00182 BC00182 V=150.0 PL=0  +MOVJ EC00178
ARCON
SFTON3D P029
SMOVL C00183 BC00183 V=11.7  +MOVJ EC00179
SMOVL C00184 BC00184 V=11.7  +MOVJ EC00180
ARCOF
SMOVL C00185 BC00185 V=800.0  +MOVJ EC00181
SMOVL C00186 BC00186 V=1000.0  +MOVJ EC00182
SFTOF3D
'EndPath W4876
MOVJ C00187 BC00187 VJ=100.00  +MOVJ EC00183 VJ=100.00
MOVJ C00188 BC00188 VJ=100.00  +MOVJ EC00184 VJ=100.00
MOVJ C00189 BC00189 VJ=100.00  +MOVJ EC00185 VJ=100.00
'Path W4877
SFTOF3D
SFTON3D P030
MOVJ C00190 BC00190 VJ=100.00  +MOVJ EC00186 VJ=100.00
SMOVL C00191 BC00191 V=800.0  +MOVJ EC00187
SMOVL C00192 BC00192 V=150.0 PL=0  +MOVJ EC00188
ARCON
SMOVL C00193 BC00193 V=10.8  +MOVJ EC00189
SMOVL C00194 BC00194 V=10.8  +MOVJ EC00190
SMOVL C00195 BC00195 V=10.0  +MOVJ EC00191
ARCOF
SMOVL C00196 BC00196 V=800.0  +MOVJ EC00192
SMOVL C00197 BC00197 V=1000.0  +MOVJ EC00193
SFTOF3D
'EndPath W4877
MOVJ C00198 BC00198 VJ=100.00  +MOVJ EC00194 VJ=100.00
MOVJ C00199 BC00199 VJ=100.00  +MOVJ EC00195 VJ=100.00
'Path W4878
SFTOF3D
SFTON3D P031
MOVJ C00200 BC00200 VJ=100.00  +MOVJ EC00196 VJ=100.00
SMOVL C00201 BC00201 V=800.0  +MOVJ EC00197
MACRO1 MJ#(0) ARGF9
SMOVL C00202 BC00202 V=150.0 PL=0  +MOVJ EC00198
ARCON
SMOVL C00203 BC00203 V=10.0 PL=0  +MOVJ EC00199
ARCON
SWVON WEV#(101)
SMOVL C00204 BC00204 V=8.3  +MOVJ EC00200
SMOVL C00205 BC00205 V=8.3  +MOVJ EC00201
SWVOF
SFTON3D P030
MACRO1 MJ#(0) ARGF14
SMOVL C00206 BC00206 V=10.0  +MOVJ EC00202
ARCOF
SMOVL C00207 BC00207 V=800.0  +MOVJ EC00203
SMOVL C00208 BC00208 V=1000.0  +MOVJ EC00204
SFTOF3D
'EndPath W4878
MOVJ C00209 BC00209 VJ=100.00  +MOVJ EC00205 VJ=100.00
MOVJ C00210 BC00210 VJ=100.00  +MOVJ EC00206 VJ=100.00
MOVJ C00211 BC00211 VJ=100.00  +MOVJ EC00207 VJ=100.00
SFTON3D P045
MACRO1 MJ#(0) ARGF6
SMOVL C00212 BC00212 V=166.7  +MOVJ EC00208
ARCON
SMOVL C00213 BC00213 V=10.0  +MOVJ EC00209
ARCOF
SMOVL C00214 BC00214 V=166.7  +MOVJ EC00210
SMOVL C00215 BC00215 V=166.7  +MOVJ EC00211
SMOVL C00216 BC00216 V=166.7  +MOVJ EC00212
ARCON
SMOVL C00217 BC00217 V=11.7  +MOVJ EC00213
ARCOF
SMOVL C00218 BC00218 V=250.0  +MOVJ EC00214
MOVJ C00219 BC00219 VJ=100.00  +MOVJ EC00215 VJ=100.00
MOVJ C00220 BC00220 VJ=100.00  +MOVJ EC00216 VJ=100.00
MOVJ C00221 BC00221 VJ=100.00  +MOVJ EC00217 VJ=100.00
SMOVL C00222 BC00222 V=166.7  +MOVJ EC00218
ARCON
SMOVL C00223 BC00223 V=11.7  +MOVJ EC00219
ARCOF
SMOVL C00224 BC00224 V=800.0  +MOVJ EC00220
SFTOF3D
MOVJ C00225 BC00225 VJ=100.00  +MOVJ EC00221 VJ=100.00
MOVJ C00226 BC00226 VJ=100.00  +MOVJ EC00222 VJ=100.00
MOVJ C00227 BC00227 VJ=100.00  +MOVJ EC00223 VJ=100.00
MOVJ C00228 BC00228 VJ=100.00  +MOVJ EC00224 VJ=100.00
MOVJ C00229 BC00229 VJ=100.00  +MOVJ EC00225 VJ=100.00
CALL JOB:CLEAN-R1_KM_NEW
'
'
'
'
'
'
'Path S4829
SFTOF3D
MOVJ C00230 BC00230 VJ=100.00  +MOVJ EC00226 VJ=100.00
MOVL C00231 BC00231 V=666.7  +MOVJ EC00227 VJ=100.00
SMOVL C00232 BC00232 V=166.7  +MOVJ EC00228
SREFP 3 C00233 BC00233  +REFP EC00229
CALL JOB:SEARCH-R1-S13D
SET P031 P006
SFTON3D P031
SMOVL C00234 BC00234 V=166.7  +MOVJ EC00230
SREFP 3 C00235 BC00235  +REFP EC00231
CALL JOB:SEARCH-R1-S13D
SET P031 P006
SFTON3D P031
SMOVL C00236 BC00236 V=166.7  +MOVJ EC00232
SMOVL C00237 BC00237 V=666.7  +MOVJ EC00233
SMOVL C00238 BC00238 V=166.7  +MOVJ EC00234
SREFP 3 C00239 BC00239  +REFP EC00235
CALL JOB:SEARCH-R1-S13D
SET P031 P006
SFTON3D P031
SMOVL C00240 BC00240 V=166.7  +MOVJ EC00236
'EndPath S4829
MOVJ C00241 BC00241 VJ=100.00  +MOVJ EC00237 VJ=100.00
'Path S4830
SFTOF3D
MOVJ C00242 BC00242 VJ=100.00  +MOVJ EC00238 VJ=100.00
SMOVL C00243 BC00243 V=666.7  +MOVJ EC00239
SMOVL C00244 BC00244 V=166.7  +MOVJ EC00240
SREFP 3 C00245 BC00245  +REFP EC00241
CALL JOB:SEARCH-R1-S13D
SET P030 P006
SFTON3D P030
SMOVL C00246 BC00246 V=166.7  +MOVJ EC00242
SMOVL C00247 BC00247 V=666.7  +MOVJ EC00243
SMOVL C00248 BC00248 V=166.7  +MOVJ EC00244
SREFP 3 C00249 BC00249  +REFP EC00245
CALL JOB:SEARCH-R1-S13D
SET P030 P006
SFTON3D P030
SMOVL C00250 BC00250 V=250.0  +MOVJ EC00246
MOVL C00251 BC00251 V=1000.0  +MOVJ EC00247 VJ=100.00
'EndPath S4830
'Path S4831
SFTOF3D
MOVJ C00252 BC00252 VJ=100.00  +MOVJ EC00248 VJ=100.00
SMOVL C00253 BC00253 V=666.7  +MOVJ EC00249
SMOVL C00254 BC00254 V=166.7  +MOVJ EC00250
SREFP 3 C00255 BC00255  +REFP EC00251
CALL JOB:SEARCH-R1-S13D
SET P029 P006
SFTON3D P029
SMOVL C00256 BC00256 V=166.7  +MOVJ EC00252
SMOVL C00257 BC00257 V=666.7  +MOVJ EC00253
SMOVL C00258 BC00258 V=166.7  +MOVJ EC00254
SREFP 3 C00259 BC00259  +REFP EC00255
CALL JOB:SEARCH-R1-S13D
SET P029 P006
SFTON3D P029
SMOVL C00260 BC00260 V=250.0  +MOVJ EC00256
MOVL C00261 BC00261 V=1000.0  +MOVJ EC00257 VJ=100.00
'EndPath S4831
'Path S4832
SFTOF3D
SMOVL C00262 BC00262 V=1200.0  +MOVJ EC00258
SMOVL C00263 BC00263 V=1000.0  +MOVJ EC00259
SMOVL C00264 BC00264 V=166.7  +MOVJ EC00260
SREFP 3 C00265 BC00265  +REFP EC00261
CALL JOB:SEARCH-R1-S13D
SET P045 P006
SFTON3D P045
SMOVL C00266 BC00266 V=166.7  +MOVJ EC00262
SMOVL C00267 BC00267 V=333.3  +MOVJ EC00263
SMOVL C00268 BC00268 V=166.7  +MOVJ EC00264
SREFP 3 C00269 BC00269  +REFP EC00265
CALL JOB:SEARCH-R1-S13D
SET P045 P006
SFTON3D P045
SMOVL C00270 BC00270 V=166.7  +MOVJ EC00266
SMOVL C00271 BC00271 V=800.0  +MOVJ EC00267
SMOVL C00272 BC00272 V=166.7  +MOVJ EC00268
SREFP 3 C00273 BC00273  +REFP EC00269
CALL JOB:SEARCH-R1-S13D
SET P045 P006
SFTON3D P045
SMOVL C00274 BC00274 V=166.7  +MOVJ EC00270
SFTOF3D
SMOVL C00275 BC00275 V=1000.0  +MOVJ EC00271
SMOVL C00276 BC00276 V=1200.0  +MOVJ EC00272
SMOVL C00277 BC00277 V=666.7  +MOVJ EC00273
SMOVL C00278 BC00278 V=166.7  +MOVJ EC00274
SREFP 3 C00279 BC00279  +REFP EC00275
CALL JOB:SEARCH-R1-S13D
SET P028 P006
SFTON3D P028
SMOVL C00280 BC00280 V=166.7  +MOVJ EC00276
SMOVL C00281 BC00281 V=666.7  +MOVJ EC00277
SMOVL C00282 BC00282 V=166.7  +MOVJ EC00278
SREFP 3 C00283 BC00283  +REFP EC00279
CALL JOB:SEARCH-R1-S13D
SET P028 P006
SFTON3D P028
SMOVL C00284 BC00284 V=166.7  +MOVJ EC00280
MOVL C00285 BC00285 V=1000.0  +MOVJ EC00281 VJ=100.00
'EndPath S4832
MOVJ C00286 BC00286 VJ=100.00  +MOVJ EC00282 VJ=100.00
'Path S4833
SFTOF3D
MOVJ C00287 BC00287 VJ=100.00  +MOVJ EC00283 VJ=100.00
MOVL C00288 BC00288 V=666.7  +MOVJ EC00284 VJ=100.00
SMOVL C00289 BC00289 V=166.7  +MOVJ EC00285
SREFP 3 C00290 BC00290  +REFP EC00286
CALL JOB:SEARCH-R1-S13D
SET P027 P006
SFTON3D P027
SMOVL C00291 BC00291 V=166.7  +MOVJ EC00287
SMOVL C00292 BC00292 V=166.7  +MOVJ EC00288
SREFP 3 C00293 BC00293  +REFP EC00289
CALL JOB:SEARCH-R1-S13D
SET P027 P006
SFTON3D P027
SMOVL C00294 BC00294 V=166.7  +MOVJ EC00290
MOVL C00295 BC00295 V=1000.0  +MOVJ EC00291 VJ=100.00
'EndPath S4833
'Path S4834
SFTOF3D
MOVJ C00296 BC00296 VJ=100.00  +MOVJ EC00292 VJ=100.00
MOVL C00297 BC00297 V=666.7  +MOVJ EC00293 VJ=100.00
SMOVL C00298 BC00298 V=166.7  +MOVJ EC00294
SREFP 3 C00299 BC00299  +REFP EC00295
CALL JOB:SEARCH-R1-S13D
SET P026 P006
SFTON3D P026
SMOVL C00300 BC00300 V=166.7  +MOVJ EC00296
SMOVL C00301 BC00301 V=166.7  +MOVJ EC00297
SREFP 3 C00302 BC00302  +REFP EC00298
CALL JOB:SEARCH-R1-S13D
SET P026 P006
SFTON3D P026
SMOVL C00303 BC00303 V=166.7  +MOVJ EC00299
'EndPath S4834
'Path S4835
SFTOF3D
MOVJ C00304 BC00304 VJ=100.00  +MOVJ EC00300 VJ=100.00
MOVL C00305 BC00305 V=666.7  +MOVJ EC00301 VJ=100.00
SMOVL C00306 BC00306 V=166.7  +MOVJ EC00302
SREFP 3 C00307 BC00307  +REFP EC00303
CALL JOB:SEARCH-R1-S13D
SET P025 P006
SFTON3D P025
SMOVL C00308 BC00308 V=166.7  +MOVJ EC00304
SMOVL C00309 BC00309 V=166.7  +MOVJ EC00305
SREFP 3 C00310 BC00310  +REFP EC00306
CALL JOB:SEARCH-R1-S13D
SET P025 P006
SFTON3D P025
SMOVL C00311 BC00311 V=166.7  +MOVJ EC00307
MOVL C00312 BC00312 V=1000.0  +MOVJ EC00308 VJ=100.00
'EndPath S4835
MOVJ C00313 BC00313 VJ=100.00  +MOVJ EC00309 VJ=100.00
MOVJ C00314 BC00314 VJ=100.00  +MOVJ EC00310 VJ=100.00
'Path S4836 (for W4841)
SFTOF3D
MOVJ C00315 BC00315 VJ=100.00  +MOVJ EC00311 VJ=100.00
MOVL C00316 BC00316 V=666.7  +MOVJ EC00312 VJ=100.00
SMOVL C00317 BC00317 V=166.7  +MOVJ EC00313
SREFP 3 C00318 BC00318  +REFP EC00314
CALL JOB:SEARCH-R1-S13D
SET P024 P006
SFTON3D P024
SMOVL C00319 BC00319 V=166.7  +MOVJ EC00315
SREFP 3 C00320 BC00320  +REFP EC00316
CALL JOB:SEARCH-R1-S13D
SET P024 P006
SFTON3D P024
SMOVL C00321 BC00321 V=166.7  +MOVJ EC00317
MOVL C00322 BC00322 V=1000.0  +MOVJ EC00318 VJ=100.00
'EndPath S4836 (for W4841)
'Path S4837 (for W4841)
SFTOF3D
MOVJ C00323 BC00323 VJ=100.00  +MOVJ EC00319 VJ=100.00
MOVL C00324 BC00324 V=666.7  +MOVJ EC00320 VJ=100.00
SMOVL C00325 BC00325 V=166.7  +MOVJ EC00321
SREFP 3 C00326 BC00326  +REFP EC00322
CALL JOB:SEARCH-R1-S13D
SET P023 P006
SFTON3D P023
SMOVL C00327 BC00327 V=166.7  +MOVJ EC00323
SREFP 3 C00328 BC00328  +REFP EC00324
CALL JOB:SEARCH-R1-S13D
SET P023 P006
SFTON3D P023
SMOVL C00329 BC00329 V=166.7  +MOVJ EC00325
MOVL C00330 BC00330 V=1000.0  +MOVJ EC00326 VJ=100.00
'EndPath S4837 (for W4841)
MOVJ C00331 BC00331 VJ=100.00  +MOVJ EC00327 VJ=100.00
MOVJ C00332 BC00332 VJ=100.00  +MOVJ EC00328 VJ=100.00
MOVJ C00333 BC00333 VJ=100.00  +MOVJ EC00329 VJ=100.00
MOVJ C00334 BC00334 VJ=100.00  +MOVJ EC00330 VJ=100.00
'Path S4838 (for W4840)
SFTOF3D
MOVJ C00335 BC00335 VJ=100.00  +MOVJ EC00331 VJ=100.00
MOVL C00336 BC00336 V=666.7  +MOVJ EC00332 VJ=100.00
SMOVL C00337 BC00337 V=166.7  +MOVJ EC00333
SREFP 3 C00338 BC00338  +REFP EC00334
CALL JOB:SEARCH-R1-S13D
SET P021 P006
SFTON3D P021
SMOVL C00339 BC00339 V=166.7  +MOVJ EC00335
SREFP 3 C00340 BC00340  +REFP EC00336
CALL JOB:SEARCH-R1-S13D
SET P021 P006
SFTON3D P021
SMOVL C00341 BC00341 V=166.7  +MOVJ EC00337
MOVL C00342 BC00342 V=1000.0  +MOVJ EC00338 VJ=100.00
'EndPath S4838 (for W4840)
MOVJ C00343 BC00343 VJ=100.00  +MOVJ EC00339 VJ=100.00
'Path S4839 (for W4840)
SFTOF3D
MOVJ C00344 BC00344 VJ=100.00  +MOVJ EC00340 VJ=100.00
MOVL C00345 BC00345 V=666.7  +MOVJ EC00341 VJ=100.00
SMOVL C00346 BC00346 V=166.7  +MOVJ EC00342
SREFP 3 C00347 BC00347  +REFP EC00343
CALL JOB:SEARCH-R1-S13D
SET P022 P006
SFTON3D P022
SMOVL C00348 BC00348 V=166.7  +MOVJ EC00344
SREFP 3 C00349 BC00349  +REFP EC00345
CALL JOB:SEARCH-R1-S13D
SET P022 P006
SFTON3D P022
SMOVL C00350 BC00350 V=166.7  +MOVJ EC00346
'EndPath S4839 (for W4840)
'Path W4840
SFTOF3D
SFTON3D P022
SMOVL C00351 BC00351 V=800.0  +MOVJ EC00347
SREFP 1 C00352 BC00352  +REFP EC00348
SREFP 2 C00353 BC00353  +REFP EC00349
SMOVL C00354 BC00354 V=150.0 PL=0  +MOVJ EC00350
MACRO1 MJ#(0) ARGF21
ARCON
SWVON WEV#(100)
SFTON3D P021
SMOVL C00355 BC00355 V=8.3  +MOVJ EC00351
ARCOF
SWVOF
SMOVL C00356 BC00356 V=800.0  +MOVJ EC00352
SMOVL C00357 BC00357 V=1000.0  +MOVJ EC00353
SFTOF3D
'EndPath W4840
MOVJ C00358 BC00358 VJ=100.00  +MOVJ EC00354 VJ=100.00
MOVJ C00359 BC00359 VJ=100.00  +MOVJ EC00355 VJ=100.00
MOVJ C00360 BC00360 VJ=100.00  +MOVJ EC00356 VJ=100.00
MOVJ C00361 BC00361 VJ=100.00  +MOVJ EC00357 VJ=100.00
'Path W4841
SFTOF3D
SFTON3D P024
MOVJ C00362 BC00362 VJ=100.00  +MOVJ EC00358 VJ=100.00
SMOVL C00363 BC00363 V=800.0  +MOVJ EC00359
SMOVL C00364 BC00364 V=150.0 PL=0  +MOVJ EC00360
ARCON
SWVON WEV#(100)
SFTON3D P023
SMOVL C00365 BC00365 V=8.3  +MOVJ EC00361
ARCOF
SWVOF
SMOVL C00366 BC00366 V=800.0  +MOVJ EC00362
SMOVL C00367 BC00367 V=1000.0  +MOVJ EC00363
SFTOF3D
'EndPath W4841
'
MOVJ C00368 BC00368 VJ=100.00  +MOVJ EC00364 VJ=100.00
'Path W4842
SFTOF3D
SFTON3D P027
MOVJ C00369 BC00369 VJ=100.00  +MOVJ EC00365 VJ=100.00
SMOVL C00370 BC00370 V=800.0  +MOVJ EC00366
SMOVL C00371 BC00371 V=150.0 PL=0  +MOVJ EC00367
MACRO1 MJ#(0) ARGF14
ARCON
SMOVL C00372 BC00372 V=10.8  +MOVJ EC00368
SMOVL C00373 BC00373 V=10.8  +MOVJ EC00369
SFTON3D P026
SMOVL C00374 BC00374 V=10.8  +MOVJ EC00370
SFTON3D P025
SMOVL C00375 BC00375 V=10.8  +MOVJ EC00371
MOVL C00376 BC00376 V=10.8  +MOVJ EC00372 VJ=0.78
ARCOF
SMOVL C00377 BC00377 V=800.0  +MOVJ EC00373
SMOVL C00378 BC00378 V=1000.0  +MOVJ EC00374
SFTOF3D
COMM SFTON3D P025
COMM MOVJ C00379 BC00379 VJ=100.00  +MOVJ EC00375 VJ=100.00
COMM SMOVL C00380 BC00380 V=800.0  +MOVJ EC00376
COMM SMOVL C00381 BC00381 V=150.0 PL=0  +MOVJ EC00377
COMM MACRO1 MJ#(0) ARGF9
COMM ARCON
COMM SMOVL C00382 BC00382 V=12.5  +MOVJ EC00378
COMM ARCOF
COMM SMOVL C00383 BC00383 V=800.0  +MOVJ EC00379
COMM SMOVL C00384 BC00384 V=1000.0  +MOVJ EC00380
COMM SFTOF3D
COMM 'EndPath W4842
COMM 'Path W4843
COMM SFTOF3D
COMM SFTON3D P026
COMM MOVJ C00385 BC00385 VJ=100.00  +MOVJ EC00381 VJ=100.00
COMM SMOVL C00386 BC00386 V=800.0  +MOVJ EC00382
COMM SMOVL C00387 BC00387 V=150.0 PL=0  +MOVJ EC00383
COMM ARCON
COMM SMOVL C00388 BC00388 V=12.5  +MOVJ EC00384
COMM ARCOF
COMM SMOVL C00389 BC00389 V=800.0  +MOVJ EC00385
COMM SMOVL C00390 BC00390 V=1000.0  +MOVJ EC00386
COMM SFTOF3D
COMM 'EndPath W4843
COMM 'Path W4844
COMM SFTOF3D
COMM SFTON3D P027
COMM MOVJ C00391 BC00391 VJ=100.00  +MOVJ EC00387 VJ=100.00
COMM SMOVL C00392 BC00392 V=800.0  +MOVJ EC00388
COMM SMOVL C00393 BC00393 V=150.0 PL=0  +MOVJ EC00389
COMM ARCON
COMM SMOVL C00394 BC00394 V=12.5  +MOVJ EC00390
COMM ARCOF
COMM SMOVL C00395 BC00395 V=800.0  +MOVJ EC00391
COMM SMOVL C00396 BC00396 V=1000.0  +MOVJ EC00392
COMM SFTOF3D
'EndPath W4844
'Path W4845
SFTOF3D
SFTON3D P028
MOVJ C00397 BC00397 VJ=100.00  +MOVJ EC00393 VJ=100.00
SMOVL C00398 BC00398 V=800.0  +MOVJ EC00394
SMOVL C00399 BC00399 V=150.0 PL=0  +MOVJ EC00395
MACRO1 MJ#(0) ARGF14
ARCON
SFTON3D P029
SMOVL C00400 BC00400 V=10.0  +MOVJ EC00396
SMOVL C00401 BC00401 V=10.0  +MOVJ EC00397
ARCOF
SMOVL C00402 BC00402 V=800.0  +MOVJ EC00398
SMOVL C00403 BC00403 V=1000.0  +MOVJ EC00399
SFTOF3D
'EndPath W4845
MOVJ C00404 BC00404 VJ=100.00  +MOVJ EC00400 VJ=100.00
MOVJ C00405 BC00405 VJ=100.00  +MOVJ EC00401 VJ=100.00
MOVJ C00406 BC00406 VJ=100.00  +MOVJ EC00402 VJ=100.00
'Path W4846
SFTOF3D
SFTON3D P030
MOVJ C00407 BC00407 VJ=100.00  +MOVJ EC00403 VJ=100.00
SMOVL C00408 BC00408 V=800.0  +MOVJ EC00404
SMOVL C00409 BC00409 V=150.0 PL=0  +MOVJ EC00405
ARCON
SMOVL C00410 BC00410 V=10.8  +MOVJ EC00406
SMOVL C00411 BC00411 V=10.8  +MOVJ EC00407
SMOVL C00412 BC00412 V=12.5  +MOVJ EC00408
SMOVL C00413 BC00413 V=12.5  +MOVJ EC00409
ARCOF
SMOVL C00414 BC00414 V=800.0  +MOVJ EC00410
SMOVL C00415 BC00415 V=1000.0  +MOVJ EC00411
SFTOF3D
'EndPath W4846
MOVJ C00416 BC00416 VJ=100.00  +MOVJ EC00412 VJ=100.00
MOVJ C00417 BC00417 VJ=100.00  +MOVJ EC00413 VJ=100.00
'Path W4847
SFTOF3D
SFTON3D P031
MOVJ C00418 BC00418 VJ=100.00  +MOVJ EC00414 VJ=100.00
SMOVL C00419 BC00419 V=800.0  +MOVJ EC00415
SMOVL C00420 BC00420 V=150.0 PL=0  +MOVJ EC00416
MACRO1 MJ#(0) ARGF9
ARCON
SWVON WEV#(101)
SMOVL C00421 BC00421 V=10.0 PL=0  +MOVJ EC00417
SMOVL C00422 BC00422 V=8.3  +MOVJ EC00418
SMOVL C00423 BC00423 V=8.3  +MOVJ EC00419
SWVOF
SFTON3D P030
SMOVL C00424 BC00424 V=10.0  +MOVJ EC00420
ARCOF
SMOVL C00425 BC00425 V=800.0  +MOVJ EC00421
SMOVL C00426 BC00426 V=1000.0  +MOVJ EC00422
SFTOF3D
'EndPath W4847
MOVJ C00427 BC00427 VJ=100.00  +MOVJ EC00423 VJ=100.00
MOVJ C00428 BC00428 VJ=100.00  +MOVJ EC00424 VJ=100.00
MACRO1 MJ#(0) ARGF6
MOVJ C00429 BC00429 VJ=100.00  +MOVJ EC00425 VJ=100.00
SFTON3D P045
SMOVL C00430 BC00430 V=133.3  +MOVJ EC00426
ARCON
SMOVL C00431 BC00431 V=11.7  +MOVJ EC00427
ARCOF
MOVJ C00432 BC00432 VJ=15.00  +MOVJ EC00428 VJ=100.00
MOVJ C00433 BC00433 VJ=80.00  +MOVJ EC00429 VJ=15.00
MOVJ C00434 BC00434 VJ=80.00  +MOVJ EC00430 VJ=80.00
SMOVL C00435 BC00435 V=133.3  +MOVJ EC00431
ARCON
SMOVL C00436 BC00436 V=11.7  +MOVJ EC00432
ARCOF
SMOVL C00437 BC00437 V=250.0  +MOVJ EC00433
SFTOF3D
MOVJ C00438 BC00438 VJ=80.00  +MOVJ EC00434 VJ=80.00
MOVJ C00439 BC00439 VJ=100.00  +MOVJ EC00435 VJ=100.00
END
